FUNCTION_BLOCK FB_Vision
VAR_INPUT
    bEnable         : BOOL;
    bTrigger        : BOOL;
    bAck            : BOOL;

	bFaultAck     : BOOL;

    bForceOffline   : BOOL;
    bForceReject    : BOOL;
	bForceTimeout : BOOL;

    nProductID      : DINT;
END_VAR

VAR_OUTPUT
    stResult        : ST_VisionResult;
    bOffline        : BOOL;
	bTimeout : BOOL;
END_VAR

VAR
    fbTrigger           : R_TRIG;
    fbInspectionTimer   : TON;
	fbTimeoutTimer    : TON;
	
    bInspectionActive   : BOOL := FALSE;
END_VAR


// VISION SIMULATION


// Communication state

bOffline := bForceOffline;

fbTrigger(CLK := bTrigger);


// Operator acknowledges technical vision fault

IF bFaultAck THEN
    bTimeout := FALSE;
END_IF;

// Offline camera aborts active inspection

IF bOffline THEN

    bInspectionActive := FALSE;
    stResult.bResultValid := FALSE;

END_IF;

// Camera ready

stResult.bReady :=
    bEnable
    AND NOT bOffline
    AND NOT bTimeout
    AND NOT bInspectionActive
    AND NOT stResult.bResultValid;

// Start inspection

IF fbTrigger.Q AND stResult.bReady THEN

    bInspectionActive := TRUE;

    stResult.bResultValid := FALSE;
    stResult.bPartPresent := FALSE;

END_IF;

// Simulated processing timer
//
// ForceTimeout prevents the normal result from arriving.

fbInspectionTimer(
    IN := bInspectionActive AND NOT bForceTimeout,
    PT := T#1S
);

// Maximum time allowed for inspection

fbTimeoutTimer(
    IN := bInspectionActive,
    PT := T#3S
);


stResult.bBusy := bInspectionActive;

// Successful inspection completed

IF bInspectionActive
   AND fbInspectionTimer.Q
   AND NOT bOffline THEN

    bInspectionActive := FALSE;

    stResult.bResultValid := TRUE;
    stResult.bPartPresent := TRUE;

    stResult.nProductID := nProductID;

    IF bForceReject THEN

        stResult.bPartOK := FALSE;
        stResult.nDefectCode := UINT#101;

        stResult.fWidth := 47.2;
        stResult.fHeight := 29.4;
        stResult.fAngle := 2.5;

    ELSE

        stResult.bPartOK := TRUE;
        stResult.nDefectCode := UINT#0;

        stResult.fWidth := 50.1;
        stResult.fHeight := 30.0;
        stResult.fAngle := 0.2;

    END_IF;

END_IF;

// Inspection timeout

IF bInspectionActive
   AND fbTimeoutTimer.Q THEN

    bInspectionActive := FALSE;

    bTimeout := TRUE;

    stResult.bResultValid := FALSE;
    stResult.bPartPresent := FALSE;

END_IF;

// PLC consumed valid inspection result

IF bAck AND stResult.bResultValid THEN

    stResult.bResultValid := FALSE;

END_IF;

END_FUNCTION_BLOCK

(* stored: Version 1.1.0.1, ProductVersion 3.1.4024.16
   POU FB_Vision: Id {e4784a81-76f0-4833-826c-513aa733616e}, SpecialFunc None *)
